{attribute 'GeneratedUsingTerminal: EL3356-0030-0025'}
{attribute addProperty BoxType "EL3356-0030-0025"}
{attribute addProperty Id "Start_calibrationBOOL1Disable_calibrationBOOL1Input_freezeBOOL1Sample_modeBOOL1TaraBOOL1"}
{attribute addProperty CRC "3118322687"}
{attribute addProperty Size "5"}
TYPE Ctrl_B9DDD3FF :
STRUCT
	{attribute addProperty Name "Start_calibration"}
	Start_calibration : BOOL;
	{attribute addProperty Name "Disable_calibration"}
	Disable_calibration : BOOL;
	{attribute addProperty Name "Input_freeze"}
	Input_freeze : BOOL;
	{attribute addProperty Name "Sample_mode"}
	Sample_mode : BOOL;
	{attribute addProperty Name "Tara"}
	Tara : BOOL;
END_STRUCT
END_TYPE

(* stored: Version 1.2.0.0, ProductVersion 3.1.4024.9
   DUT Ctrl_B9DDD3FF: Id {5362f820-58e9-435b-8453-b08d6be06ea9} *)
